// TIA Portal project "FBD" (V14)

(* hardware
DEVICE "S7-1200 station_1"  S7-1200 Station
   slot 0: "Rack_0"  S7-1200 Rack  Rack  V1.0
   slot 1: "PLC_1"  CPU 1214C DC/DC/DC  6ES7 214-1AG40-0XB0  V4.2
*)

// ===== PLC "PLC_1"  CPU 1214C DC/DC/DC =====

VAR_GLOBAL   // PLC tag table "Default tag table"
   "Entrada 1" AT %M100.1 : Bool;
   "Entrada 2" AT %M100.2 : Bool;
   "Entrada 3" AT %M100.3 : Bool;
   "Saida 1" AT %M100.4 : Bool;
END_VAR

FUNCTION "FDB" : Void   // FC1, FBD
{ S7_Optimized_Access := 'TRUE' }
VERSION : 0.1
BEGIN

REGION Network 1
   // FDB EXEMPLO
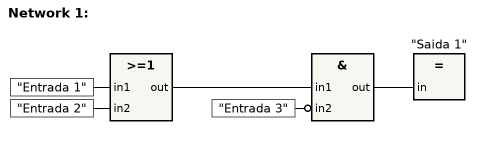
   "Saida 1" := ("Entrada 1" OR "Entrada 2") AND NOT "Entrada 3";
END_REGION
END_FUNCTION

ORGANIZATION_BLOCK "Main"   // OB1, LAD, ProgramCycle
TITLE = "Main Program Sweep (Cycle)"
{ S7_Optimized_Access := 'TRUE' }
VERSION : 0.1
   VAR_INPUT
      Initial_Call : Bool;   // Initial call of this OB
      Remanence : Bool;   // =True, if remanent data are available
   END_VAR
BEGIN

REGION Network 1
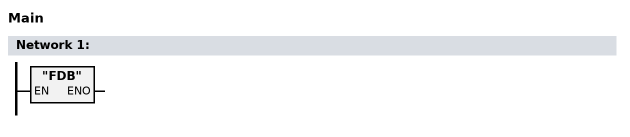
   RUNG wire#powerrail
      "FDB"()
   END_RUNG
   // the same network as SCL:
   "FDB"();
END_REGION
END_ORGANIZATION_BLOCK